(* CODESYS project test-Git

Project tree, tasks and I/O mapping:
  Device : 600L/700 (Linux), Exor International, version 3.5.16.30
    application Application
      libraries: Standard, 3.5.18.0 (System)
      task MainTask (cyclic, interval t#20ms, priority 1) calls PLC_PRG
      program PLC_PRG [ST]
*)

// Device/Application/PLC_PRG
PROGRAM PLC_PRG
VAR
END_VAR

END_PROGRAM
